// Mitsubishi GX Works2 project: goodgood (1) (1)   PLC: FX3G

// global labels: Global1
VAR_GLOBAL
  allDayOn AT Y007 : BOOL;
  petelAmount AT D1610 : REAL;
  inputPetelAmount AT D1600 : REAL;
  inputLemonAmount AT D1700 : REAL;
  lemonAmount AT D1710 : REAL;
  inputHomerAmount AT D1800 : REAL;
  homerAmount AT D1810 : REAL;
  emergencyLamp AT Y005 : BOOL;
  emergencyEnd AT X005 : BOOL;
  noValidity AT M6 : BOOL;
  endDay AT M7 : BOOL;
  begin AT X007 : BOOL;
  analogInput1 AT D8280 : INT;
  saveTypeValue AT D1900 : REAL;
  typeValue AT D1500 : REAL;
END_VAR
VAR_GLOBAL CONSTANT
  typeRagil : REAL := 5;
  typtypeRagileRagil : INT := 5;
END_VAR
VAR_GLOBAL
  pinuk AT M2 : BOOL;
END_VAR
VAR_GLOBAL CONSTANT
  const6 : REAL := 6.0;
  const10 : REAL := 10.0;
END_VAR
VAR_GLOBAL
  ragil AT M3 : BOOL;
  sample AT X001 : BOOL;
END_VAR
VAR_GLOBAL CONSTANT
  minPetelPinuk : REAL := 385.0;
  minLemonPinuk : REAL := 665.0;
  minHomerPinuk : REAL := 210.0;
END_VAR
VAR_GLOBAL
  checkValidityPinuk AT M1 : BOOL;
END_VAR
VAR_GLOBAL CONSTANT
  minPetelRagil : REAL := 280.0;
  minLemonRagil : REAL := 455.0;
END_VAR
VAR_GLOBAL
  checkValidityRagil AT M5 : BOOL;
  startMaking AT M8 : BOOL;
  making AT Y000 : BOOL;
  freezing AT X002 : BOOL;
END_VAR
VAR_GLOBAL CONSTANT
  const400 : REAL := 400.0;
END_VAR
VAR_GLOBAL
  holdTime AT M9 : BOOL;
  freezingLight AT Y002 : BOOL;
  holdRagil AT M12 : BOOL;
  helpValidityPinuk AT M13 : BOOL;
  helpValidityRagil AT M14 : BOOL;
END_VAR
VAR_GLOBAL CONSTANT
  makingRagil : INT := 840;
  const840 : INT := 840;
END_VAR
VAR_GLOBAL
  containerMakingLemon AT D1400 : REAL;
END_VAR
VAR_GLOBAL CONSTANT
  const350 : REAL := 350.0;
END_VAR
VAR_GLOBAL
  containerMakingPetel AT D2000 : REAL;
END_VAR
VAR_GLOBAL CONSTANT
  const490 : REAL := 490.0;
  const560 : REAL := 560.0;
  const700 : REAL := 700.0;
END_VAR
VAR_GLOBAL
  TC_1 AT TC1 : BOOL;
END_VAR
VAR_GLOBAL CONSTANT
  const8 : INT := 80;
END_VAR
VAR_GLOBAL
  containerFreezingLemon AT D2010 : REAL;
  containerFreezingPetel AT D1910 : REAL;
  mixing AT M15 : BOOL;
  containerMixing AT D1950 : REAL;
END_VAR
VAR_GLOBAL CONSTANT
  const28 : REAL := 28.0;
  const70 : REAL := 70.0;
END_VAR
VAR_GLOBAL
  helpFlick AT M16 : BOOL;
  TC_3 AT TC3 : BOOL;
  TC_4 AT TC4 : BOOL;
END_VAR
VAR_GLOBAL CONSTANT
  const20 : INT := 20;
END_VAR
VAR_GLOBAL
  flickering1 AT Y005 : BOOL;
  flickering2 AT Y006 : BOOL;
  TC_5 AT TC5 : BOOL;
  isTemp10 AT M17 : BOOL;
  TempSensor AT X003 : BOOL;
  TC_6 AT TC6 : BOOL;
END_VAR
VAR_GLOBAL CONSTANT
  const5sec : REAL := 5.0;
END_VAR
VAR_GLOBAL
  finishFreezingTime AT TS6 : BOOL;
END_VAR
VAR_GLOBAL CONSTANT
  const500 : REAL := 5.0;
  const300 : REAL := 3.0;
  const0 : REAL;
END_VAR
VAR_GLOBAL
  startPacking AT X004 : BOOL;
  mixingTime AT D3000 : REAL;
  isPinukMixed AT M63 : BOOL;
  isRagilMixed AT M64 : BOOL;
  TimerMixingPinuk AT TC10 : BOOL;
END_VAR
VAR_GLOBAL CONSTANT
  MixingTo5sec : INT := 50;
END_VAR
VAR_GLOBAL
  stopMixingPinuk AT TS10 : BOOL;
  FinishMixingPinukLight AT M70 : BOOL;
  TimerMixingRagil AT TC11 : BOOL;
END_VAR
VAR_GLOBAL CONSTANT
  MixingTo3sec : INT := 30;
END_VAR
VAR_GLOBAL
  stopMixingRagil AT TS11 : BOOL;
  FinishMixingRagilLight AT M71 : BOOL;
  packOneConeCounter AT CC0 : BOOL;
  packOneCone AT X000 : BOOL;
END_VAR
VAR_GLOBAL CONSTANT
  CountConeDone : INT := 1;
END_VAR
VAR_GLOBAL
  packOnePackageCounter AT CC1 : BOOL;
END_VAR
VAR_GLOBAL CONSTANT
  Count7ConesDone : INT := 7;
END_VAR
VAR_GLOBAL
  startCount AT CS0 : BOOL;
  stopCount AT CS1 : BOOL;
  start6More AT Y004 : BOOL;
  countOneIteration AT M99 : BOOL;
  amountPackages AT D1360 : REAL;
END_VAR
VAR_GLOBAL CONSTANT
  addOnePackage : REAL := 1.0;
END_VAR
VAR_GLOBAL
  mixingIsComplete AT M37 : BOOL;
END_VAR
VAR_GLOBAL CONSTANT
  const40 : REAL := 40.0;
END_VAR
VAR_GLOBAL
  outputPackages AT D1111 : REAL;
  analogOutput AT D8282 : INT;
  inputGumiAmount AT D1802 : REAL;
  GumiAmount AT D1806 : REAL;
  floatInput AT D6000 : REAL;
  bdika AT X006 : BOOL;
END_VAR
VAR_GLOBAL CONSTANT
  const5 : INT := 50;
  minHomerRagil : REAL := 105.0;
END_VAR
VAR_GLOBAL
  endMakingLight AT TS1 : BOOL;
END_VAR
VAR_GLOBAL CONSTANT
  const10Sec : INT := 10;
END_VAR
VAR_GLOBAL
  helpFlickering1 AT TS4 : BOOL;
  helpFlickering2 AT TS5 : BOOL;
  finishFreezing AT M58 : BOOL;
  holdNoVadility AT M75 : BOOL;
  resetPackageCounter AT CN1 : INT;
  helpReset AT M17 : BOOL;
  holdPinuk AT M10 : BOOL;
END_VAR

// task Task_01 (event TRUE, interval 0, priority 31): POU_01

PROGRAM POU_01
(* structured ladder/FBD written out as ST: instructions are called as NAME(EN, inputs, outputs); _pN, _eN, _tN stand for wires *)
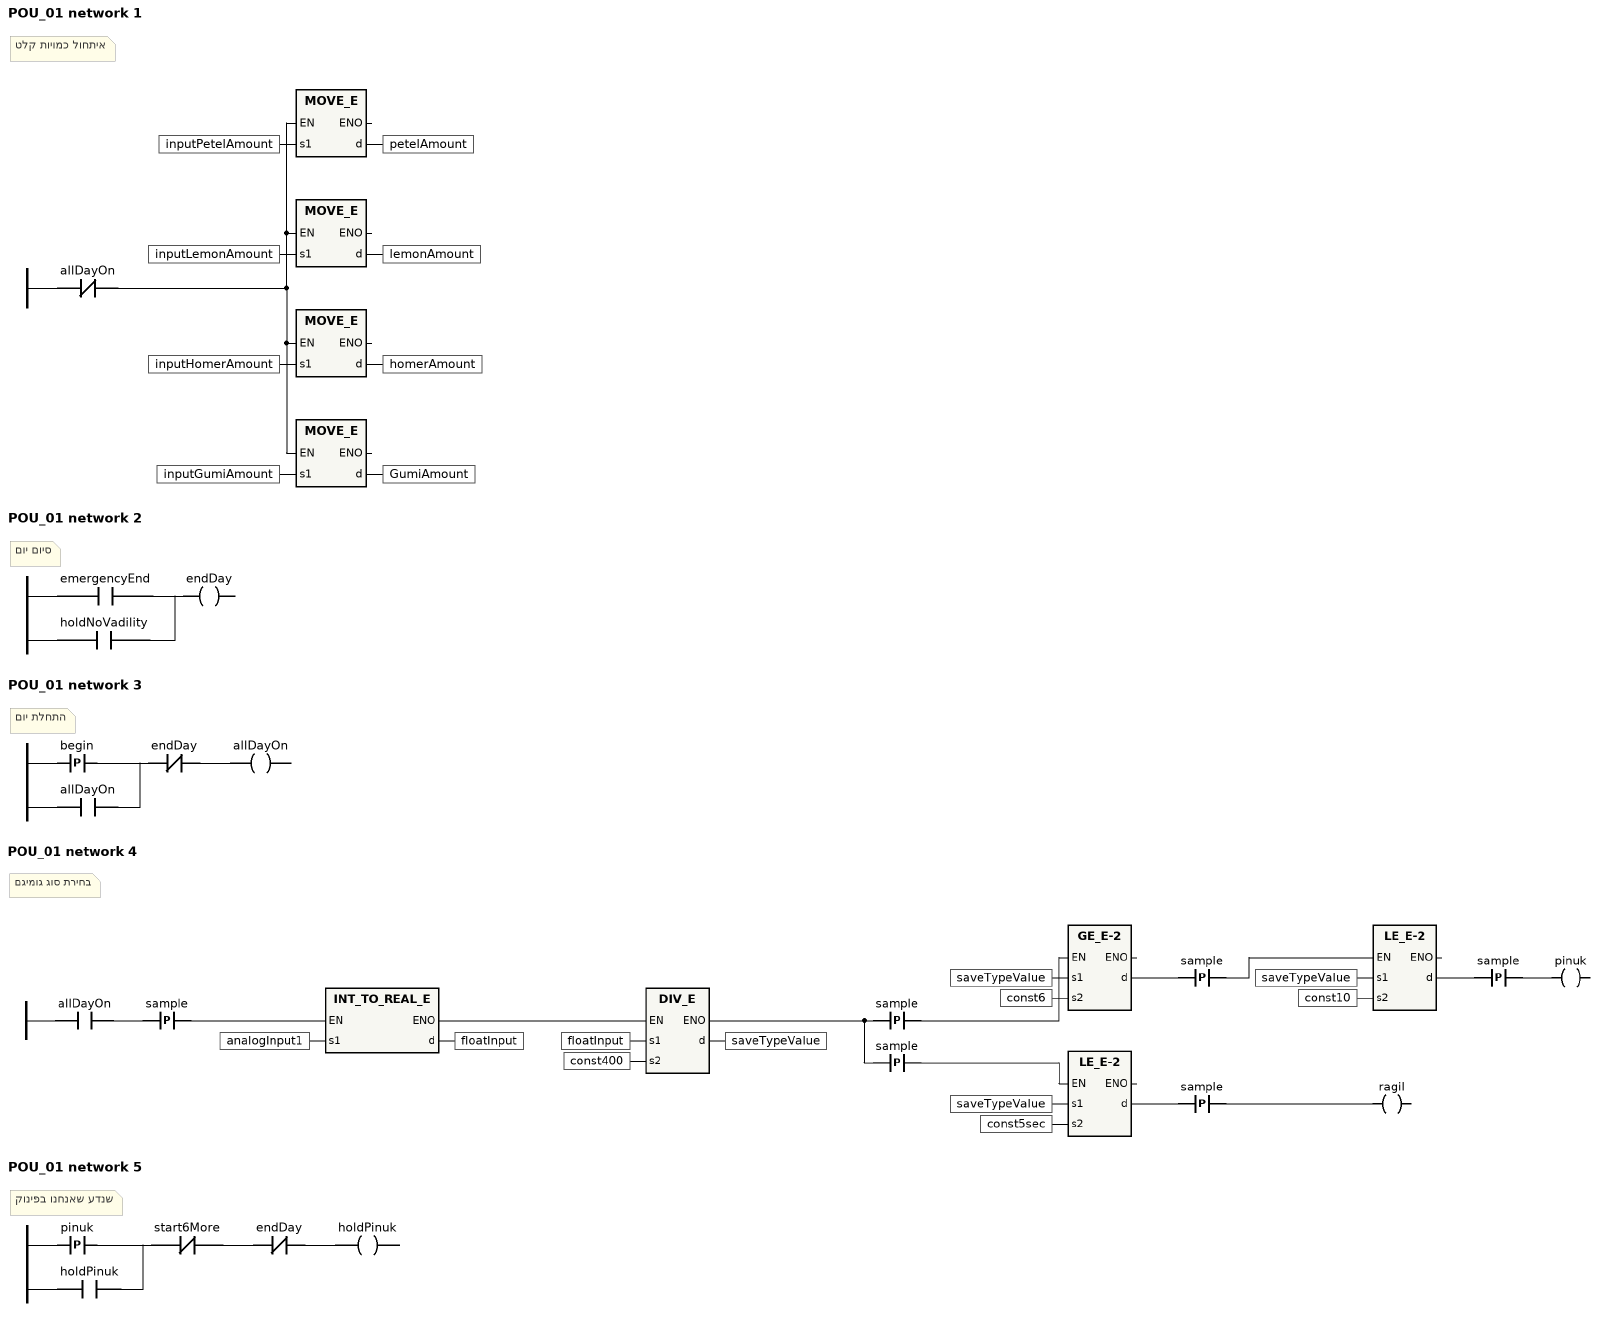
(* network 1 *)
(* איתחול כמויות קלט *)
_p1 := NOT allDayOn;
MOVE_E(_p1, inputPetelAmount, petelAmount);
MOVE_E(_p1, inputLemonAmount, lemonAmount);
MOVE_E(_p1, inputHomerAmount, homerAmount);
MOVE_E(_p1, inputGumiAmount, GumiAmount);
(* network 2 *)
(* סיום יום *)
endDay := emergencyEnd OR holdNoVadility;
(* network 3 *)
(* התחלת יום *)
allDayOn := (LDP(TRUE, begin) OR allDayOn) AND NOT endDay;
(* network 4 *)
(* בחירת סוג גומיגם *)
_e1 := INT_TO_REAL_E(allDayOn AND LDP(TRUE, sample), analogInput1, floatInput);
_e2 := DIV_E(_e1, floatInput, const400, saveTypeValue);
GE_E(_e2 AND LDP(TRUE, sample), saveTypeValue, const6, _t3);
LE_E(_t3 AND LDP(TRUE, sample), saveTypeValue, const10, _t4);
pinuk := _t4 AND LDP(TRUE, sample);
LE_E(_e2 AND LDP(TRUE, sample), saveTypeValue, const5sec, _t5);
ragil := _t5 AND LDP(TRUE, sample);
(* network 5 *)
(* שנדע שאנחנו בפינוק *)
holdPinuk := ((LDP(TRUE, pinuk) OR holdPinuk) AND NOT start6More) AND NOT endDay;
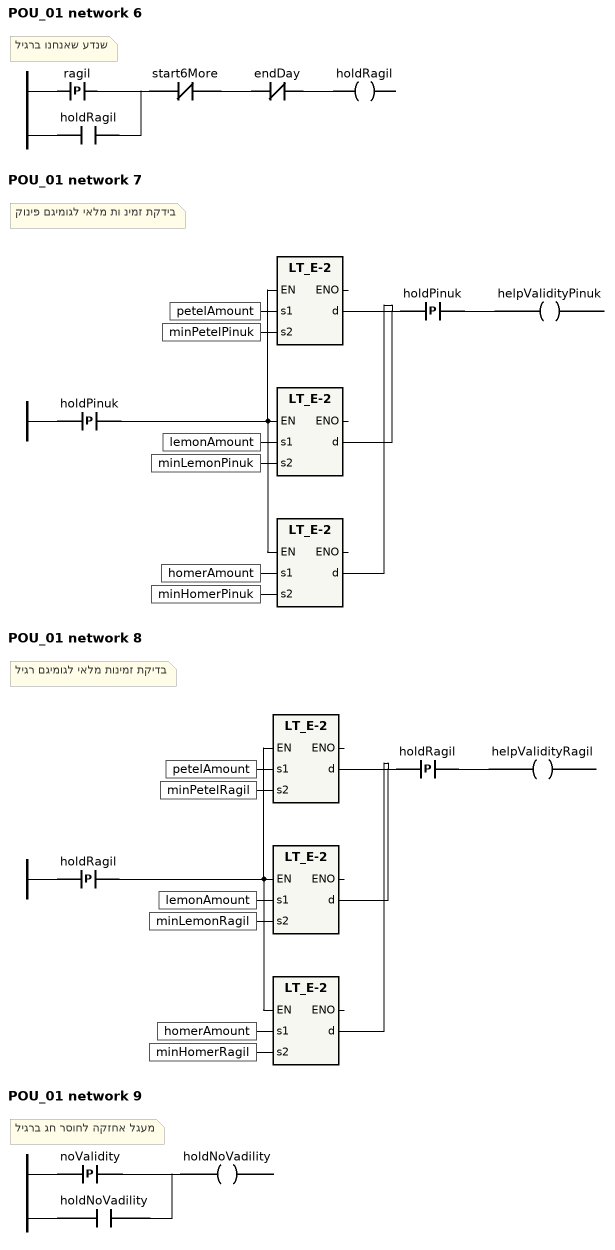
(* network 6 *)
(* שנדע שאנחנו ברגיל *)
holdRagil := ((LDP(TRUE, ragil) OR holdRagil) AND NOT start6More) AND NOT endDay;
(* network 7 *)
(* בידקת זמינ ות מלאי לגומיגם פינוק *)
_p1 := LDP(TRUE, holdPinuk);
LT_E(_p1, petelAmount, minPetelPinuk, _t2);
LT_E(_p1, lemonAmount, minLemonPinuk, _t3);
LT_E(_p1, homerAmount, minHomerPinuk, _t4);
helpValidityPinuk := (_t2 OR _t3 OR _t4) AND LDP(TRUE, holdPinuk);
(* network 8 *)
(* בדיקת זמינות מלאי לגומיגם רגיל *)
_p1 := LDP(TRUE, holdRagil);
LT_E(_p1, petelAmount, minPetelRagil, _t2);
LT_E(_p1, lemonAmount, minLemonRagil, _t3);
LT_E(_p1, homerAmount, minHomerRagil, _t4);
helpValidityRagil := (_t2 OR _t3 OR _t4) AND LDP(TRUE, holdRagil);
(* network 9 *)
(* מעגל אחזקה לחוסר חג ברגיל *)
holdNoVadility := LDP(TRUE, noValidity) OR holdNoVadility;
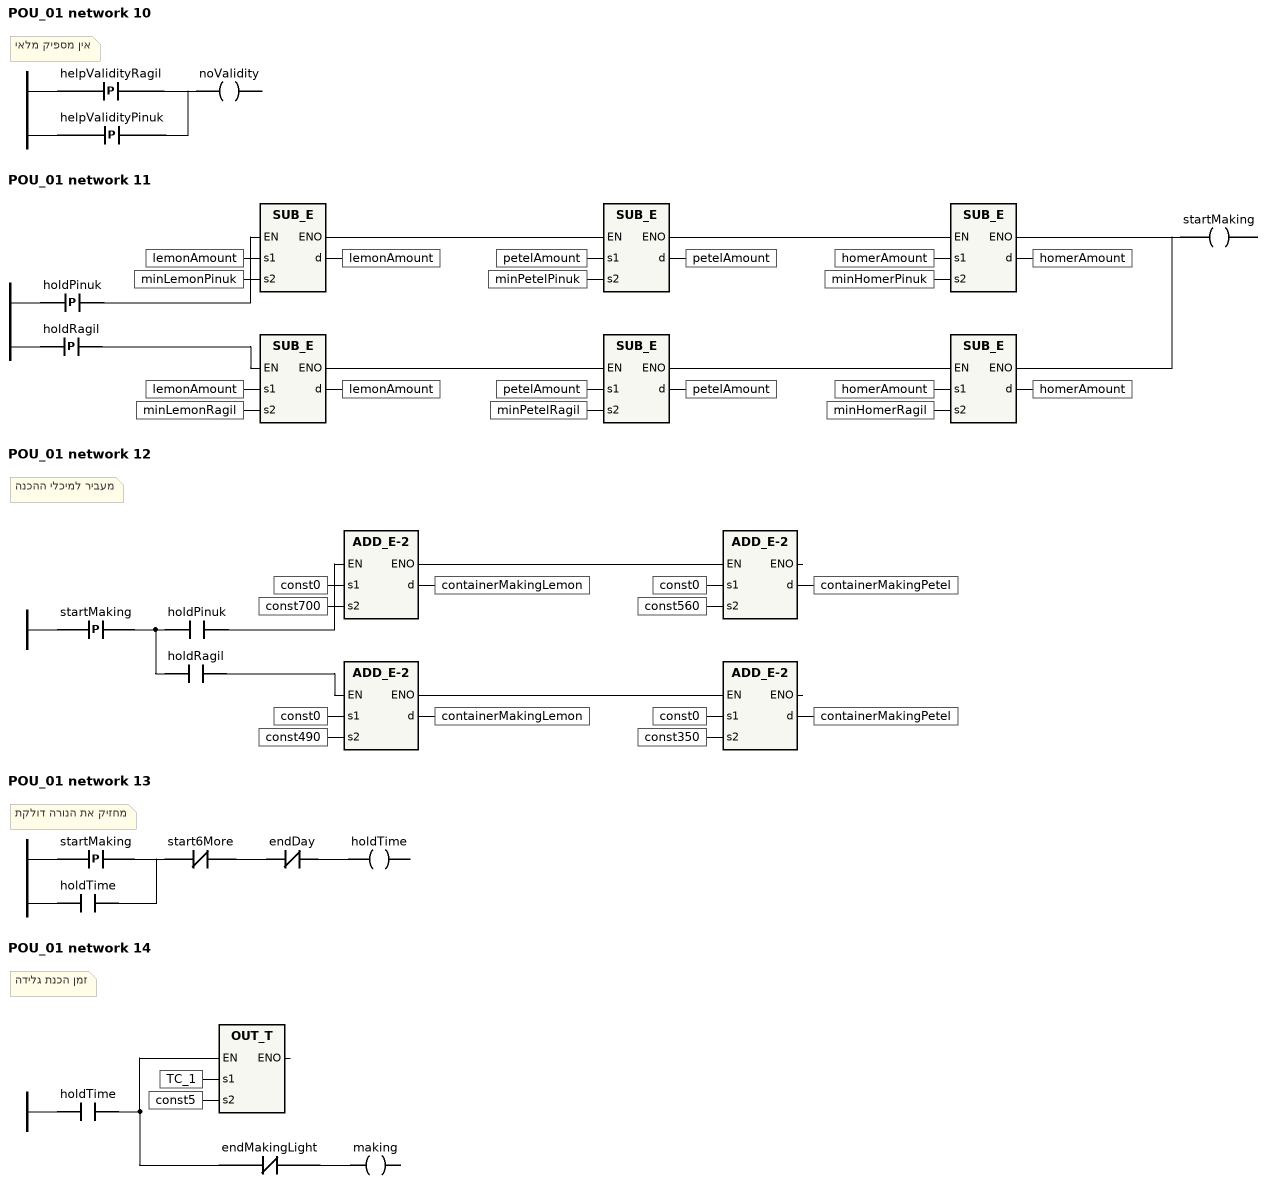
(* network 10 *)
(* אין מספיק מלאי *)
noValidity := LDP(TRUE, helpValidityRagil) OR LDP(TRUE, helpValidityPinuk);
(* network 11 *)
_e1 := SUB_E(LDP(TRUE, holdPinuk), lemonAmount, minLemonPinuk, lemonAmount);
_e2 := SUB_E(_e1, petelAmount, minPetelPinuk, petelAmount);
_e3 := SUB_E(_e2, homerAmount, minHomerPinuk, homerAmount);
_e4 := SUB_E(LDP(TRUE, holdRagil), lemonAmount, minLemonRagil, lemonAmount);
_e5 := SUB_E(_e4, petelAmount, minPetelRagil, petelAmount);
_e6 := SUB_E(_e5, homerAmount, minHomerRagil, homerAmount);
startMaking := _e3 OR _e6;
(* network 12 *)
(* מעביר למיכלי ההכנה *)
_p1 := LDP(TRUE, startMaking);
_e2 := ADD_E(_p1 AND holdPinuk, const0, const700, containerMakingLemon);
ADD_E(_e2, const0, const560, containerMakingPetel);
_e3 := ADD_E(_p1 AND holdRagil, const0, const490, containerMakingLemon);
ADD_E(_e3, const0, const350, containerMakingPetel);
(* network 13 *)
(* מחזיק את הנורה דולקת *)
holdTime := ((LDP(TRUE, startMaking) OR holdTime) AND NOT start6More) AND NOT endDay;
(* network 14 *)
(* זמן הכנת גלידה *)
OUT_T(holdTime, TC_1, const5);
making := holdTime AND NOT endMakingLight;
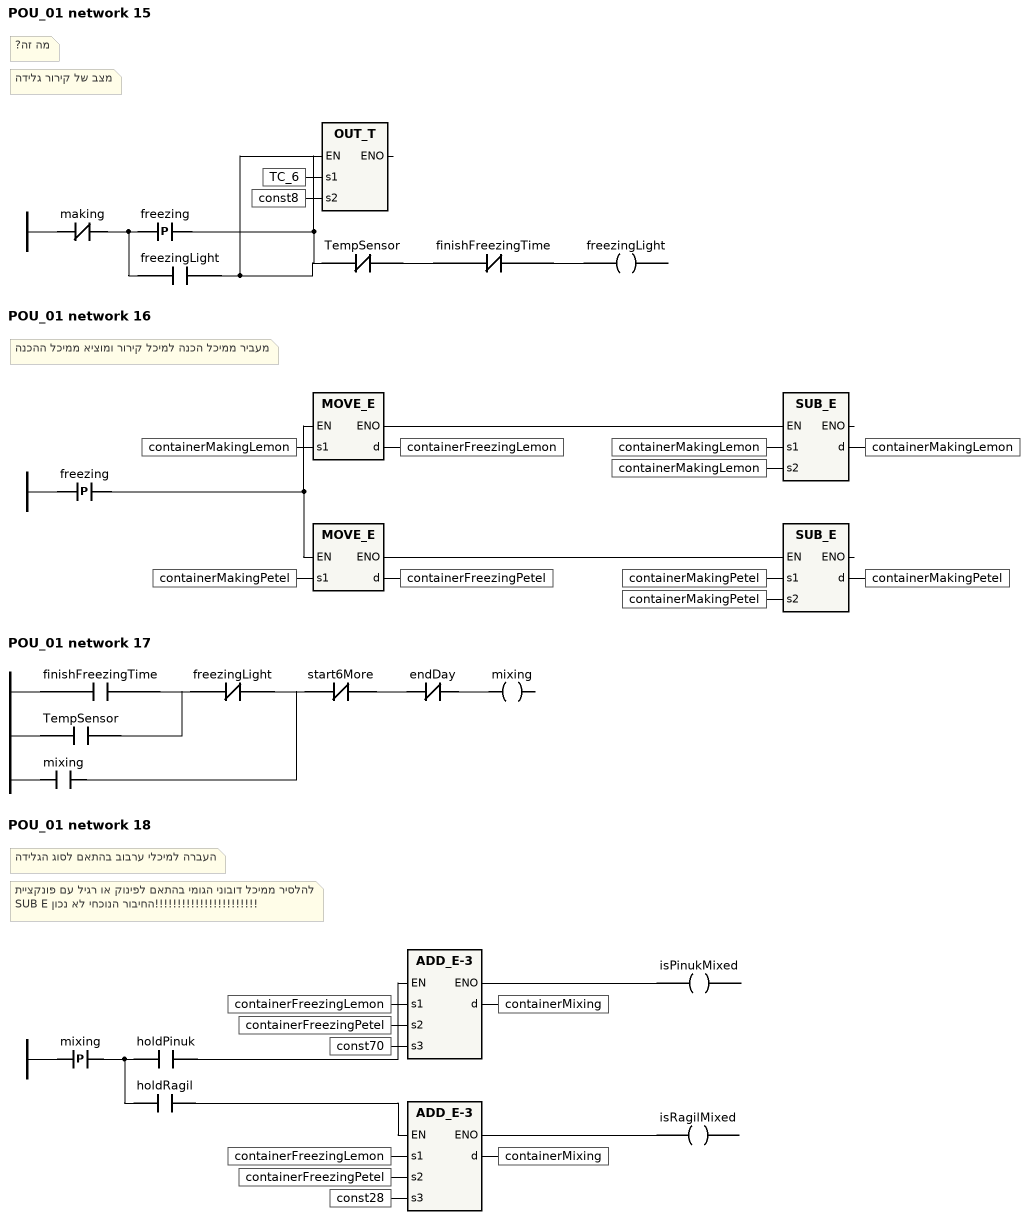
(* network 15 *)
(* מה זה? *)
(* מצב של קירור גלידה *)
_p1 := NOT making;
_p2 := (_p1 AND LDP(TRUE, freezing)) OR (_p1 AND freezingLight);
OUT_T(_p2, TC_6, const8);
freezingLight := _p2 AND NOT TempSensor AND NOT finishFreezingTime;
(* network 16 *)
(* מעביר ממיכל הכנה למיכל קירור ומוציא ממיכל ההכנה *)
_p1 := LDP(TRUE, freezing);
_e2 := MOVE_E(_p1, containerMakingLemon, containerFreezingLemon);
SUB_E(_e2, containerMakingLemon, containerMakingLemon, containerMakingLemon);
_e3 := MOVE_E(_p1, containerMakingPetel, containerFreezingPetel);
SUB_E(_e3, containerMakingPetel, containerMakingPetel, containerMakingPetel);
(* network 17 *)
mixing := ((((finishFreezingTime OR TempSensor) AND NOT freezingLight) OR mixing) AND NOT start6More) AND NOT endDay;
(* network 18 *)
(* העברה למיכלי ערבוב בהתאם לסוג הגלידה *)
(* להלסיר ממיכל דובוני הגומי בהתאם לפינוק או רגיל עם פונקציית SUB E החיבור הנוכחי לא נכון!!!!!!!!!!!!!!!!!!!!!!! *)
_p1 := LDP(TRUE, mixing);
_e2 := ADD_E(_p1 AND holdPinuk, containerFreezingLemon, containerFreezingPetel, const70, containerMixing);
isPinukMixed := _e2;
_e3 := ADD_E(_p1 AND holdRagil, containerFreezingLemon, containerFreezingPetel, const28, containerMixing);
isRagilMixed := _e3;
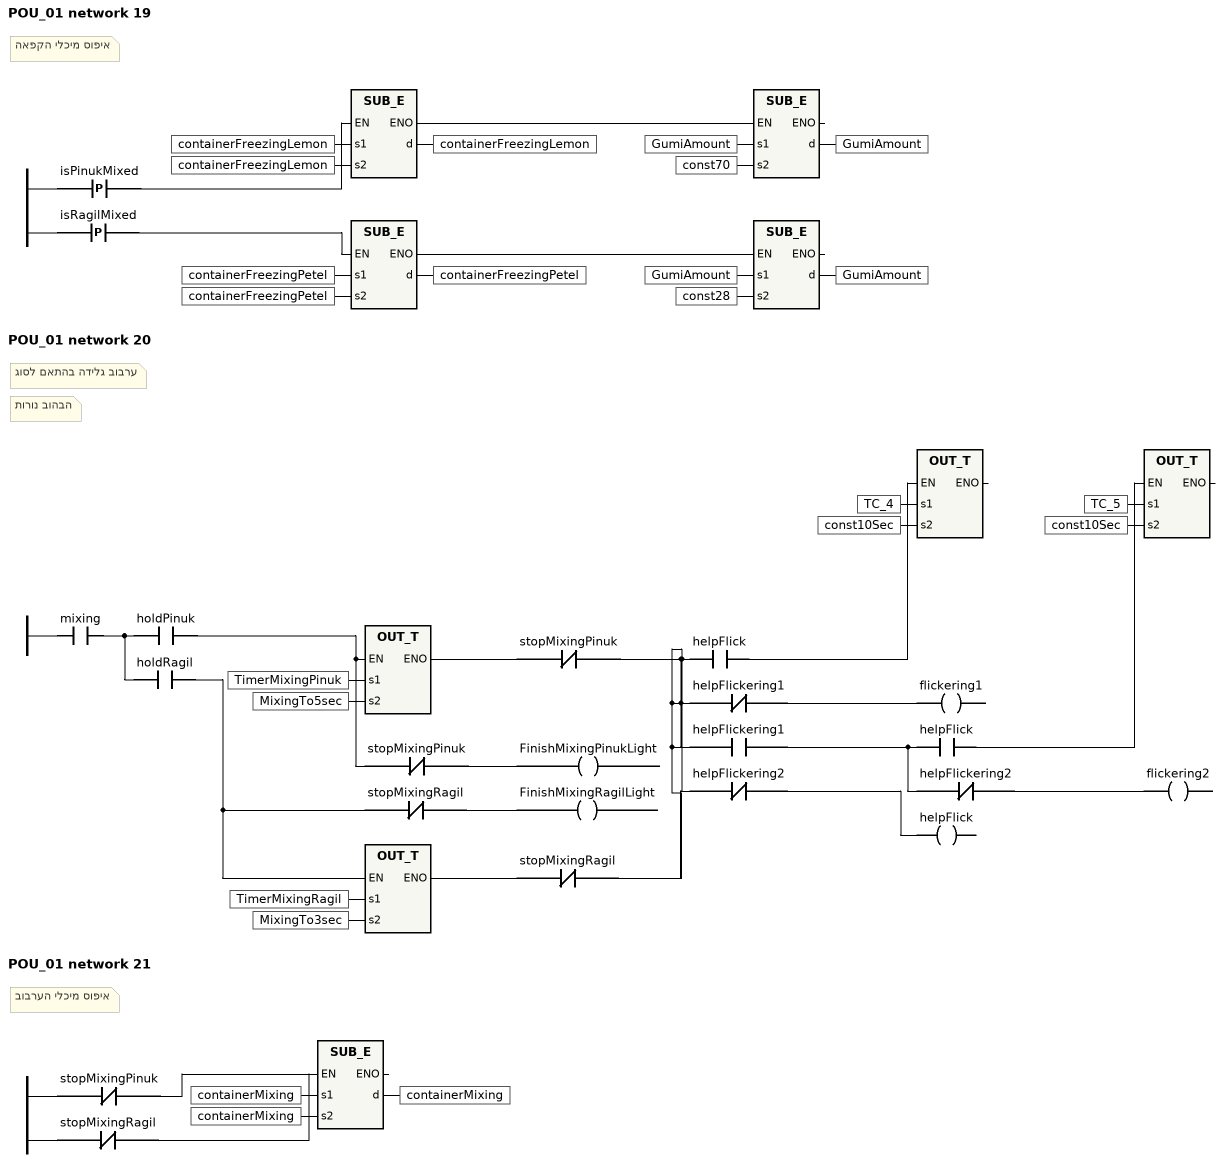
(* network 19 *)
(* איפוס מיכלי הקפאה *)
_e1 := SUB_E(LDP(TRUE, isPinukMixed), containerFreezingLemon, containerFreezingLemon, containerFreezingLemon);
SUB_E(_e1, GumiAmount, const70, GumiAmount);
_e2 := SUB_E(LDP(TRUE, isRagilMixed), containerFreezingPetel, containerFreezingPetel, containerFreezingPetel);
SUB_E(_e2, GumiAmount, const28, GumiAmount);
(* network 20 *)
(* ערבוב גלידה בהתאם לסוג *)
(* הבהוב נורות *)
_p1 := mixing AND holdPinuk;
_e2 := OUT_T(_p1, TimerMixingPinuk, MixingTo5sec);
_p3 := mixing AND holdRagil;
_e4 := OUT_T(_p3, TimerMixingRagil, MixingTo3sec);
_p5 := (_e2 AND NOT stopMixingPinuk) OR (_e4 AND NOT stopMixingRagil);
OUT_T(_p5 AND helpFlick, TC_4, const10Sec);
flickering1 := _p5 AND NOT helpFlickering1;
_p6 := _p5 AND helpFlickering1;
OUT_T(_p6 AND helpFlick, TC_5, const10Sec);
FinishMixingPinukLight := _p1 AND NOT stopMixingPinuk;
flickering2 := _p6 AND NOT helpFlickering2;
helpFlick := _p5 AND NOT helpFlickering2;
FinishMixingRagilLight := _p3 AND NOT stopMixingRagil;
(* network 21 *)
(* איפוס מיכלי הערבוב *)
SUB_E((NOT stopMixingPinuk) OR (NOT stopMixingRagil), containerMixing, containerMixing, containerMixing);
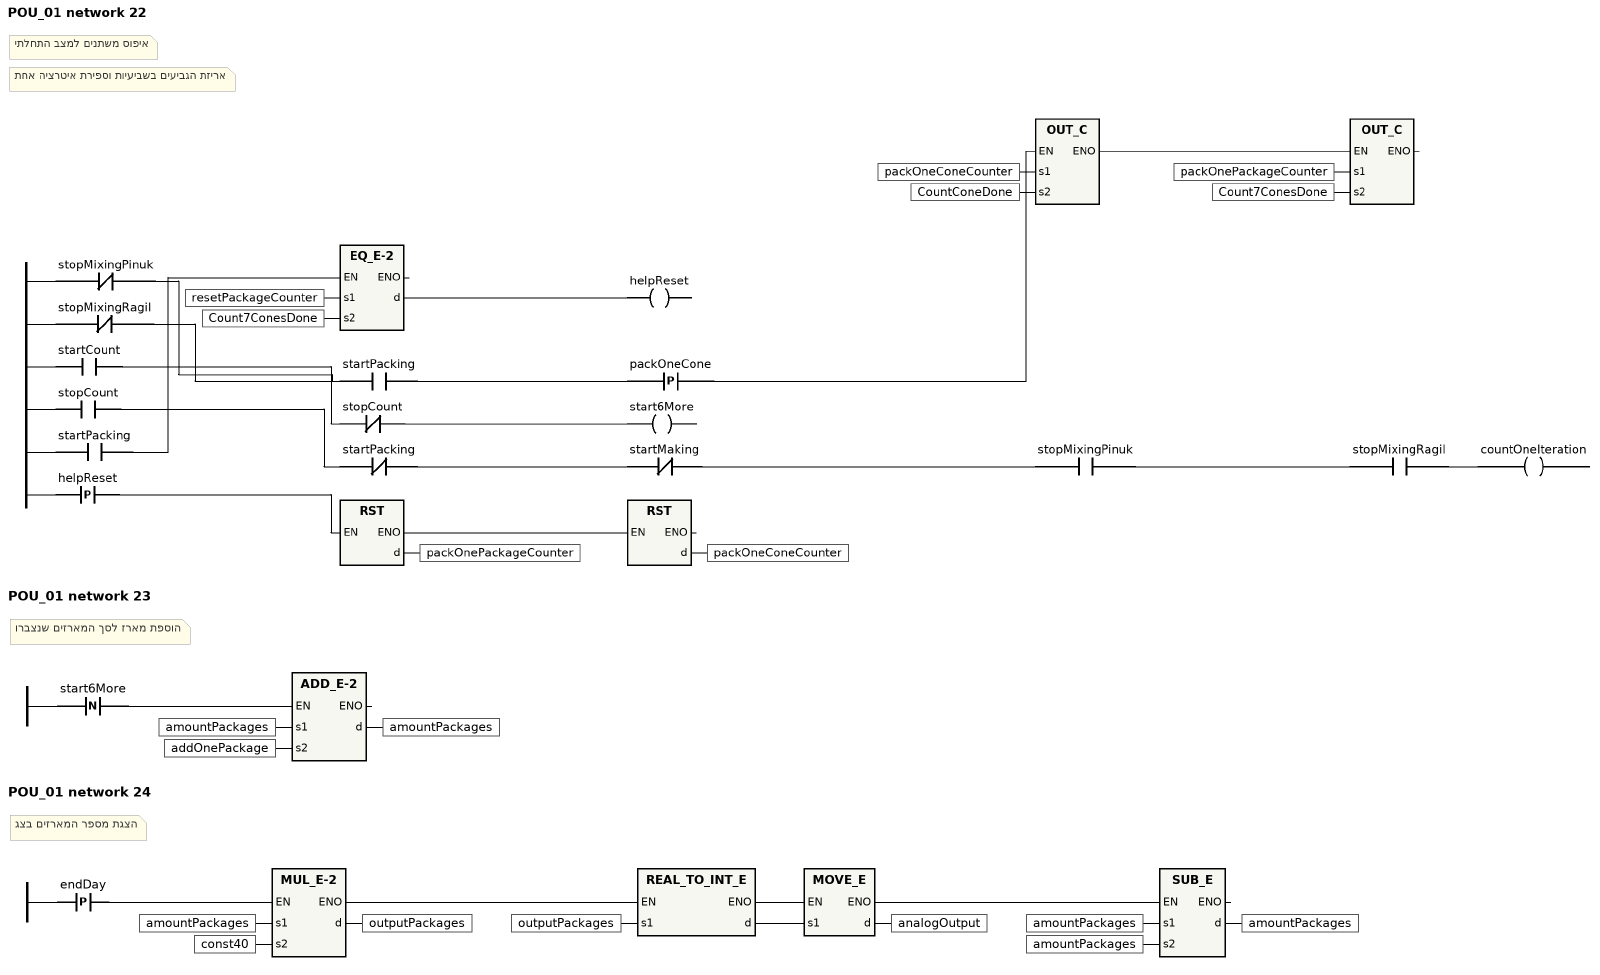
(* network 22 *)
(* איפוס משתנים למצב התחלתי *)
(* אריזת הגביעים בשביעיות וספירת איטרציה אחת *)
_e1 := OUT_C((((NOT stopMixingPinuk) OR (NOT stopMixingRagil)) AND startPacking) AND LDP(TRUE, packOneCone), packOneConeCounter, CountConeDone);
OUT_C(_e1, packOnePackageCounter, Count7ConesDone);
start6More := startCount AND NOT stopCount;
countOneIteration := stopCount AND NOT startPacking AND NOT startMaking AND stopMixingPinuk AND stopMixingRagil;
EQ_E(startPacking, resetPackageCounter, Count7ConesDone, _t2);
helpReset := _t2;
_e3 := RST(LDP(TRUE, helpReset), packOnePackageCounter);
RST(_e3, packOneConeCounter);
(* network 23 *)
(* הוספת מארז לסך המארזים שנצברו *)
ADD_E(LDF(TRUE, start6More), amountPackages, addOnePackage, amountPackages);
(* network 24 *)
(* הצגת מספר המארזים בצג *)
_e1 := MUL_E(LDP(TRUE, endDay), amountPackages, const40, outputPackages);
_e3 := REAL_TO_INT_E(_e1, outputPackages, _t2);
_e4 := MOVE_E(_e3, _t2, analogOutput);
SUB_E(_e4, amountPackages, amountPackages, amountPackages);
END_PROGRAM
